{attribute 'pack_mode' := '1'}
TYPE TManUtilities :
	STRUCT
		TAspiration				: TManButton;
		TVacuum				: TManButton;
		bPowerIsOn				: BOOL;
		bDrivesIsOn				: BOOL;
		b24VOK					: BOOL;
		b48VOK					: BOOL;
		bAirPressureOK			: BOOL;
		bMainVacuumOK			: BOOL;
		bAspirationOK			: BOOL;
		bAspirationIsOn			: BOOL;
		TResetAspirationUseTime	: TManButton;
		dwAspirationUseTime		: DWORD;
		TResetVacuumUseTime	: TManButton;
		dwVacuumUseTime		: DWORD;
	END_STRUCT
END_TYPE

(* stored: Version 1.1.0.1, ProductVersion 3.1.4022.12
   DUT TManUtilities: Id {e82ad44f-1dad-43bd-a5e7-1043a9e9b275} *)
